// TwinCAT 3 PLC project neh_tst
// ProgramVersion: 3.1.4022.7
// libraries:
//   LCLS General, * (SLAC)
//   lcls-twincat-common-components, * (SLAC)
//   lcls-twincat-motion, * (SLAC)
//   PMPS, * (SLAC - LCLS)
//   Tc2_Standard, * (Beckhoff Automation GmbH)
//   Tc2_System, * (Beckhoff Automation GmbH)
//   Tc3_Module, * (Beckhoff Automation GmbH)
// project tree:
//   / PlcTask.TcTTO
//   POUs/ MAIN.TcPOU
// real-time tasks:
//   TASK PlcTask: cycle T#10ms, priority 20, ADS port 350
// motion (NC):
// I/O:
//   DEVICE Device 1 (EtherCAT), AmsNetId 172.21.148.90.2.1
//     Term 6 (EK1200) [EK1200-5000 EtherCAT Power supply (2A E-Bus)]
//       Term 3 (EL3002) [EL3002 2Ch. Ana. Input +/-10V]
//       Term 8 (EK1122) [EK1122 2 port EtherCAT junction]
//         Term 9 (EK1100) [EK1100 EtherCAT Coupler (2A E-Bus)]
//           Term 10 (EL7041)
//           Term 11 (EL5042) [EL5042 2Ch. BiSS-C Encoder]
//           Term 12 (EL2004)
//           Term 13 (EL3314) [EL3314 4Ch. Ana. Input Thermocouple (TC)]
//           Term 14 (EL3052) [EL3052 2Ch. Ana. Input 4-20mA]
//           Term 15 (EL3062) [EL3062 2Ch. Ana. Input 0-10V]
//           Term 16 (EL4004) [EL4004 4Ch. Ana. Output 0-10V, 12bit]
//           Term 17 (EL9011)
// variable links:
//   neh_tst Instance <-> Device 1 (EtherCAT)/Term 6 (EK1200)/Term 3 (EL3002)
//     PlcTask Inputs/MAIN.rawValidatorVoltage <-> AI Standard Channel 1/Value
//   neh_tst Instance <-> Device 1 (EtherCAT)/Term 6 (EK1200)/Term 8 (EK1122)/Term 9 (EK1100)/Term 10 (EL7041)
//     PlcTask Inputs/MAIN.M1.bLimitBackwardEnable <-> STM Status/Status/Digital input 2
//     PlcTask Inputs/MAIN.M1.bLimitForwardEnable <-> STM Status/Status/Digital input 1
//   neh_tst Instance <-> Device 1 (EtherCAT)/Term 6 (EK1200)/Term 8 (EK1122)/Term 9 (EK1100)/Term 11 (EL5042)
//     PlcTask Inputs/MAIN.M1.nRawEncoderULINT <-> FB Inputs Channel 1/Position
//   neh_tst Instance <-> Device 1 (EtherCAT)/Term 6 (EK1200)/Term 8 (EK1122)/Term 9 (EK1100)/Term 12 (EL2004)
//     PlcTask Outputs/MAIN.M1.bBrakeRelease <-> Channel 1/Output
//   neh_tst Instance <-> Device 1 (EtherCAT)/Term 6 (EK1200)/Term 8 (EK1122)/Term 9 (EK1100)/Term 15 (EL3062)
//     PlcTask Inputs/MAIN.fbPowerMeter.iVoltageINT <-> AI Standard Channel 1/Value
//   neh_tst Instance <-> NC-Task 1 SAF/Axes/Axis 1
//     PlcTask Inputs/MAIN.M1.Axis.NcToPlc <-> Outputs/ToPlc
//     PlcTask Outputs/MAIN.M1.Axis.PlcToNc <-> Inputs/FromPlc

CONFIGURATION neh_tst
    RESOURCE PLC ON TwinCAT3
        TASK PlcTask(INTERVAL := T#10ms, PRIORITY := 20);
        PROGRAM MAIN WITH PlcTask : MAIN;
    END_RESOURCE
END_CONFIGURATION

// ---- POUs/MAIN.TcPOU
PROGRAM MAIN
VAR
    (* control flow bool*)
    bInit: BOOL;

    // Y motor (state select).
    fbYStage: FB_MotionStage;

    (* state maintenence *)
    fbStateDefaults: FB_PositionState_Defaults;

    {attribute 'pytmc' := '
        pv: MMS
        astPositionState.array: 1..4
    '}
    fbStates: FB_PositionStatePMPS1D;
    astPositionState: ARRAY[1..GeneralConstants.MAX_STATES] OF ST_PositionState;
    fbArrCheckWrite: FB_CheckPositionStateWrite;

    stOut: ST_PositionState;
    // Settings for the POWERMETER state.
    stPower: ST_PositionState;
    // Settings for the YAG1 state.
    stYag1: ST_PositionState;
    // Settings for the YAG2 state.
    stYag2: ST_PositionState;

    // The fast fault output to fault to.
    fbFFHWO: FB_HardwareFFOutput;
    // The arbiter to request beam conditions from.
    fbArbiter: FB_Arbiter(1);

    {attribute 'pytmc' := '
        pv: MMS:STATE:SET
        io: io
    '}
    eEnumSet: E_PPM_States;
    // Set this to TRUE to enable input state moves, or FALSE to disable them.
    bEnableMotion: BOOL;
    // Set this to TRUE to enable beam parameter checks, or FALSE to disable them.
    bEnableBeamParams: BOOL;
    // Set this to TRUE to enable position limit checks, or FALSE to disable them.
    bEnablePositionLimits: BOOL;
    // The name of the device for use in the PMPS DB lookup and diagnostic screens.
    sDeviceName: STRING;
    // The name of the transition state in the PMPS database.
    sTransitionKey: STRING;
    // Set this to TRUE to re-read the loaded database immediately (useful for debug).
    bReadDBNow: BOOL;

    {attribute 'pytmc' := 'pv: NEH:PPM
                           io: i'}
    {attribute 'TcLinkTo' := '.iVoltageINT := TIIB[Term 15 (EL3062)]^AI Standard Channel 1^Value'}
    fbPowerMeter: FB_PPM_PowerMeter;

    {attribute 'TcLinkTo' := 'TIIB[Term 3 (EL3002)]^AI Standard Channel 1^Value'}
	rawValidatorVoltage AT %I*: INT;    
	
    fValidatorVoltage : LREAL;
	
	{attribute 'TcLinkTo' := 'TIIB[Term 3 (EL3002)]^AI Inputs Channel 2^Value'}
	rVVV AT %I* : DINT;
	fVVV : LREAL;

    // IM1K3-PPM: 1 Axis
    {attribute 'TcLinkTo' := '.bLimitForwardEnable  := TIIB[Term 10 (EL7041)]^STM Status^Status^Digital input 1;
                              .bLimitBackwardEnable := TIIB[Term 10 (EL7041)]^STM Status^Status^Digital input 2;
                              .bBrakeRelease        := TIIB[Term 12 (EL2004)]^Channel 1^Output;
                              .nRawEncoderULINT     := TIIB[Term 11 (EL5042)]^FB Inputs Channel 1^Position'}
    {attribute 'pytmc' := 'pv: NEH:PPM:MMS'}
    M1: ST_MotionStage := (sName := 'NEH:PPM:MMS', nEnableMode := ENUM_StageEnableMode.ALWAYS, bPowerSelf := TRUE, bHardwareEnable := True);
    iVoltageINT: INT;
	
	
	fbGetPMVoltage: FB_AnalogInput;
	fVoltageOther : LREAL;
END_VAR
VAR CONSTANT
    // State defaults if not provided
    fDelta: LREAL := 2;
    fAccel: LREAL := 200;
    fOutDecel: LREAL := 25;
END_VAR
VAR_OUTPUT
    // The current position state as an enum.
    {attribute 'pytmc' := '
        pv: MMS:STATE:GET
        io: i
    '}
    eEnumGet: E_PPM_States;
    // The PMPS database lookup associated with the current position state.
    stDbStateParams: ST_DbStateParams;
END_VAR

IF NOT bInit THEN
    bInit := TRUE;

	// normal op
    //M1.nEnableMode := ENUM_StageEnableMode.DURING_MOTION;
    
	//M1.nEnableMode := ENUM_StageEnableMode.ALWAYS;
    //M1.bHardwareEnable := TRUE;
	//M1.bPowerSelf := TRUE;
    // Partial backcompat, this used to set fVelocity too but this should be set per install
    (*fbStateDefaults(stPositionState:=stOut, sNameDefault:='OUT', fDeltaDefault:=fDelta, fAccelDefault:=fAccel, fDecelDefault:=fOutDecel);
    fbStateDefaults(stPositionState:=stPower, sNameDefault:='POWERMETER', fDeltaDefault:=fDelta, fAccelDefault:=fAccel, fDecelDefault:=fAccel);
    fbStateDefaults(stPositionState:=stYag1, sNameDefault:='YAG1', fDeltaDefault:=fDelta, fAccelDefault:=fAccel, fDecelDefault:=fAccel);
    fbStateDefaults(stPositionState:=stYag2, sNameDefault:='YAG2', fDeltaDefault:=fDelta, fAccelDefault:=fAccel, fDecelDefault:=fAccel);*)
END_IF

fbYStage(stMotionStage:=M1);
(*
// We need to update from PLC or from EPICS, but not both
fbArrCheckWrite(
    astPositionState:=astPositionState,
    bCheck:=TRUE,
    bSave:=FALSE,
);
IF NOT fbArrCheckWrite.bHadWrite THEN
    astPositionState[E_PPM_States.OUT] := stOut;
    astPositionState[E_PPM_States.POWERMETER] := stPower;
    astPositionState[E_PPM_States.YAG1] := stYag1;
    astPositionState[E_PPM_States.YAG2] := stYag2;
END_IF

fbStates(
    stMotionStage:=M1,
    astPositionState:=astPositionState,
    eEnumSet:=eEnumSet,
    eEnumGet:=eEnumGet,
    fbFFHWO:=fbFFHWO,
    fbArbiter:=fbArbiter,
    bEnableMotion:=bEnableMotion,
    bEnableBeamParams:=bEnableBeamParams,
    bEnablePositionLimits:=bEnablePositionLimits,
    sDeviceName:=sDeviceName,
    sTransitionKey:=sTransitionKey,
    bReadDBNow:=bReadDBNow,
    stDbStateParams=>stDbStateParams,
);

fbArrCheckWrite(
    astPositionState:=astPositionState,
    bCheck:=FALSE,
    bSave:=TRUE,
);

stOut := astPositionState[E_PPM_States.OUT];
stPower := astPositionState[E_PPM_States.POWERMETER];
stYag1 := astPositionState[E_PPM_States.YAG1];
stYag2 := astPositionState[E_PPM_States.YAG2];
*)
fbPowerMeter();


fValidatorVoltage := rawValidatorVoltage / EXPT(2, 12) * 10;

(*
rVVV := rVVV AND 16#7FFFFF;
fVVV := rVVV / EXPT(2,23) * 5;
*)

fbGetPMVoltage(
    iRaw := rawValidatorVoltage,
    iTermBits := 15,
    fTermMax := 10000,
    fTermMin := 0,
    fReal => fVoltageOther);

END_PROGRAM
